ABB RAPID module: Module1.mod

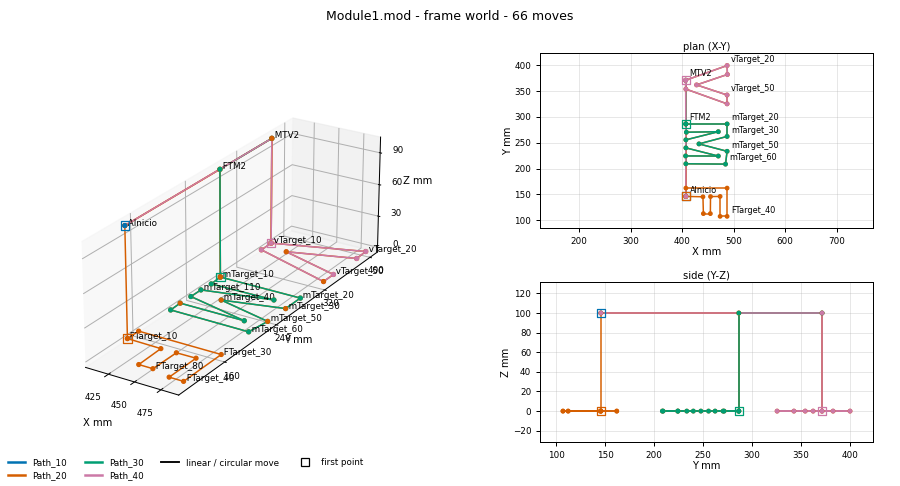
[picture p0: tool path of Module1.mod in frame world, 66 of 68 moves have a stored position in this frame; points joined in program order, loops and branches not executed]
MODULE Module1
	CONST robtarget AInicio:=[[0,-225.593,-100],[1,0,0,0],[0,0,0,0],[9E+09,9E+09,9E+09,9E+09,9E+09,9E+09]];
	CONST robtarget FTarget_10:=[[0,-225.593,0],[1,0,0,0],[0,0,0,0],[9E+09,9E+09,9E+09,9E+09,9E+09,9E+09]];
	CONST robtarget FTarget_20:=[[0,-209.44,0],[1,0,0,0],[0,0,0,0],[9E+09,9E+09,9E+09,9E+09,9E+09,9E+09]];
	CONST robtarget FTarget_30:=[[-80,-209.44,0],[1,0,0,0],[0,0,0,0],[9E+09,9E+09,9E+09,9E+09,9E+09,9E+09]];
	CONST robtarget FTarget_40:=[[-80,-264.284,0],[1,0,0,0],[0,0,0,0],[9E+09,9E+09,9E+09,9E+09,9E+09,9E+09]];
	CONST robtarget FTarget_50:=[[-66.466,-264.284,0],[1,0,0,0],[0,0,0,0],[9E+09,9E+09,9E+09,9E+09,9E+09,9E+09]];
	CONST robtarget FTarget_60:=[[-66.466,-225.593,0],[1,0,0,0],[0,0,0,0],[9E+09,9E+09,9E+09,9E+09,9E+09,9E+09]];
	CONST robtarget FTarget_70:=[[-47.849,-225.879,0],[1,0,0,0],[0,0,0,0],[9E+09,9E+09,9E+09,9E+09,9E+09,9E+09]];
	CONST robtarget FTarget_80:=[[-47.53,-258.99,0],[1,0,0,0],[0,0,0,0],[9E+09,9E+09,9E+09,9E+09,9E+09,9E+09]];
	CONST robtarget FTarget_90:=[[-33.997,-258.99,0],[1,0,0,0],[0,0,0,0],[9E+09,9E+09,9E+09,9E+09,9E+09,9E+09]];
	CONST robtarget FTarget_100:=[[-33.164,-226.306,0],[1,0,0,0],[0,0,0,0],[9E+09,9E+09,9E+09,9E+09,9E+09,9E+09]];
	CONST robtarget FTarget_110:=[[0,-225.593,0],[1,0,0,0],[0,0,0,0],[9E+09,9E+09,9E+09,9E+09,9E+09,9E+09]];
	CONST robtarget FTM1:=[[0,-225.593,-100],[1,0,0,0],[0,0,0,0],[9E+09,9E+09,9E+09,9E+09,9E+09,9E+09]];
	CONST robtarget FTM2:=[[0,-84.966,-100],[1,0,0,0],[0,0,0,0],[9E+09,9E+09,9E+09,9E+09,9E+09,9E+09]];
	CONST robtarget mTarget_10:=[[0,-84.966,0],[1,0,0,0],[0,0,0,0],[9E+09,9E+09,9E+09,9E+09,9E+09,9E+09]];
	CONST robtarget mTarget_20:=[[-80,-84.966,0],[1,0,0,0],[0,0,0,0],[9E+09,9E+09,9E+09,9E+09,9E+09,9E+09]];
	CONST robtarget mTarget_30:=[[-80,-109.14,0],[1,0,0,0],[0,0,0,0],[9E+09,9E+09,9E+09,9E+09,9E+09,9E+09]];
	CONST robtarget mTarget_40:=[[-25.429,-123.656,0],[1,0,0,0],[0,0,0,0],[9E+09,9E+09,9E+09,9E+09,9E+09,9E+09]];
	CONST robtarget mTarget_50:=[[-80,-138.008,0],[1,0,0,0],[0,0,0,0],[9E+09,9E+09,9E+09,9E+09,9E+09,9E+09]];
	CONST robtarget mTarget_60:=[[-76.954,-162.904,0],[1,0,0,0],[0,0,0,0],[9E+09,9E+09,9E+09,9E+09,9E+09,9E+09]];
	CONST robtarget mTarget_70:=[[0,-162.237,0],[1,0,0,0],[0,0,0,0],[9E+09,9E+09,9E+09,9E+09,9E+09,9E+09]];
	CONST robtarget mTarget_80:=[[0.53,-147.013,0],[1,0,0,0],[0,0,0,0],[9E+09,9E+09,9E+09,9E+09,9E+09,9E+09]];
	CONST robtarget mTarget_90:=[[-62.974,-147.23,0],[1,0,0,0],[0,0,0,0],[9E+09,9E+09,9E+09,9E+09,9E+09,9E+09]];
	CONST robtarget mTarget_100:=[[0,-131.35,0],[1,0,0,0],[0,0,0,0],[9E+09,9E+09,9E+09,9E+09,9E+09,9E+09]];
	CONST robtarget mTarget_110:=[[0,-115.798,0],[1,0,0,0],[0,0,0,0],[9E+09,9E+09,9E+09,9E+09,9E+09,9E+09]];
	CONST robtarget mTarget_120:=[[-62.974,-99.973,0],[1,0,0,0],[0,0,0,0],[9E+09,9E+09,9E+09,9E+09,9E+09,9E+09]];
	CONST robtarget mTarget_130:=[[-0.986,-101.003,0],[1,0,0,0],[0,0,0,0],[9E+09,9E+09,9E+09,9E+09,9E+09,9E+09]];
	CONST robtarget mTarget_140:=[[0,-84.966,0],[1,0,0,0],[0,0,0,0],[9E+09,9E+09,9E+09,9E+09,9E+09,9E+09]];
	CONST robtarget MTV1:=[[0,-84.966,-100],[1,0,0,0],[0,0,0,0],[9E+09,9E+09,9E+09,9E+09,9E+09,9E+09]];
	CONST robtarget MTV2:=[[0.326,-0.089,-100],[1,0,0,0],[0,0,0,0],[9E+09,9E+09,9E+09,9E+09,9E+09,9E+09]];
	CONST robtarget vTarget_10:=[[0.326,-0.089,0],[1,0,0,0],[0,0,0,0],[9E+09,9E+09,9E+09,9E+09,9E+09,9E+09]];
	CONST robtarget vTarget_20:=[[-80.066,28.469,0],[1,0,0,0],[0,0,0,0],[9E+09,9E+09,9E+09,9E+09,9E+09,9E+09]];
	CONST robtarget vTarget_30:=[[-80.616,11.146,0],[1,0,0,0],[0,0,0,0],[9E+09,9E+09,9E+09,9E+09,9E+09,9E+09]];
	CONST robtarget vTarget_40:=[[-20.791,-9.168,0],[1,0,0,0],[0,0,0,0],[9E+09,9E+09,9E+09,9E+09,9E+09,9E+09]];
	CONST robtarget vTarget_50:=[[-80,-28.758,0],[1,0,0,0],[0,0,0,0],[9E+09,9E+09,9E+09,9E+09,9E+09,9E+09]];
	CONST robtarget vTarget_60:=[[-80,-45.893,0],[1,0,0,0],[0,0,0,0],[9E+09,9E+09,9E+09,9E+09,9E+09,9E+09]];
	CONST robtarget vTarget_70:=[[0,-17.244,0],[1,0,0,0],[0,0,0,0],[9E+09,9E+09,9E+09,9E+09,9E+09,9E+09]];
	CONST robtarget vTarget_80:=[[0.326,-0.089,0],[1,0,0,0],[0,0,0,0],[9E+09,9E+09,9E+09,9E+09,9E+09,9E+09]];
	CONST robtarget vTarget_80_final:=[[0.326,-0.089,-100],[1,0,0,0],[0,0,0,0],[9E+09,9E+09,9E+09,9E+09,9E+09,9E+09]];
	CONST robtarget ZInicio:=[[0,-225.593,-100],[1,0,0,0],[0,0,0,0],[9E+09,9E+09,9E+09,9E+09,9E+09,9E+09]];
	CONST jointtarget HomePosition:=[[0,0,0,0,0,0],[9E+09,9E+09,9E+09,9E+09,9E+09,9E+09]];
	CONST jointtarget ChangeTool:=[[90.000002504,24.671787339,-34.427722191,-0.000016273,9.755934852,0.000016038],[9E+09,9E+09,9E+09,9E+09,9E+09,9E+09]];
    !***********************************************************
    !
    ! Módulo:  Module1
    !
    ! Descripción:
    !   <Introduzca la descripción aquí>
    !
    ! Autor: Administrador
    !
    ! Versión: 1.0
    !
    !***********************************************************


    !***********************************************************
    !
    ! Procedimiento Main
    !
    !   Este es el punto de entrada de su programa
    !
    !***********************************************************
    PROC main()
		Home1;
		WaitDI EntDI_1,1;
		SetDO SalDO_1,1;
		Path_10;
		Path_20;
		Home1;
		WaitDI EntDI_2,1;
		ToolChange;
		SetDO SalDO_1,0;
        !Añada aquí su código
    ENDPROC
	PROC Path_10()
	    MoveJ AInicio,v100,z10,Tooldata_MARCADOR\WObj:=Workobject_INICIALES;
	ENDPROC
	PROC Path_20()
	    MoveL FTarget_10,v100,z10,Tooldata_MARCADOR\WObj:=Workobject_INICIALES;
	    MoveL FTarget_20,v100,z10,Tooldata_MARCADOR\WObj:=Workobject_INICIALES;
	    MoveL FTarget_30,v100,z10,Tooldata_MARCADOR\WObj:=Workobject_INICIALES;
	    MoveL FTarget_40,v100,z10,Tooldata_MARCADOR\WObj:=Workobject_INICIALES;
	    MoveL FTarget_50,v100,z10,Tooldata_MARCADOR\WObj:=Workobject_INICIALES;
	    MoveL FTarget_60,v100,z10,Tooldata_MARCADOR\WObj:=Workobject_INICIALES;
	    MoveL FTarget_70,v100,z10,Tooldata_MARCADOR\WObj:=Workobject_INICIALES;
	    MoveL FTarget_80,v100,z10,Tooldata_MARCADOR\WObj:=Workobject_INICIALES;
	    MoveL FTarget_90,v100,z10,Tooldata_MARCADOR\WObj:=Workobject_INICIALES;
	    MoveL FTarget_100,v100,z10,Tooldata_MARCADOR\WObj:=Workobject_INICIALES;
	    MoveL FTarget_110,v100,z10,Tooldata_MARCADOR\WObj:=Workobject_INICIALES;
	    MoveL FTM1,v100,z10,Tooldata_MARCADOR\WObj:=Workobject_INICIALES;
	    MoveL FTM2,v100,z10,Tooldata_MARCADOR\WObj:=Workobject_INICIALES;
		MoveL mTarget_10,v100,z10,Tooldata_MARCADOR\WObj:=Workobject_INICIALES;
		MoveL mTarget_20,v100,z10,Tooldata_MARCADOR\WObj:=Workobject_INICIALES;
		MoveL mTarget_30,v100,z10,Tooldata_MARCADOR\WObj:=Workobject_INICIALES;
		MoveL mTarget_40,v100,z10,Tooldata_MARCADOR\WObj:=Workobject_INICIALES;
		MoveL mTarget_50,v100,z10,Tooldata_MARCADOR\WObj:=Workobject_INICIALES;
		MoveL mTarget_60,v100,z10,Tooldata_MARCADOR\WObj:=Workobject_INICIALES;
		MoveL mTarget_70,v100,z10,Tooldata_MARCADOR\WObj:=Workobject_INICIALES;
		MoveL mTarget_80,v100,z10,Tooldata_MARCADOR\WObj:=Workobject_INICIALES;
		MoveL mTarget_90,v100,z10,Tooldata_MARCADOR\WObj:=Workobject_INICIALES;
		MoveL mTarget_100,v100,z10,Tooldata_MARCADOR\WObj:=Workobject_INICIALES;
		MoveL mTarget_110,v100,z10,Tooldata_MARCADOR\WObj:=Workobject_INICIALES;
		MoveL mTarget_120,v100,z10,Tooldata_MARCADOR\WObj:=Workobject_INICIALES;
		MoveL mTarget_130,v100,z10,Tooldata_MARCADOR\WObj:=Workobject_INICIALES;
		MoveL mTarget_140,v100,z10,Tooldata_MARCADOR\WObj:=Workobject_INICIALES;
		MoveL MTV1,v100,z10,Tooldata_MARCADOR\WObj:=Workobject_INICIALES;
		MoveL MTV2,v100,z10,Tooldata_MARCADOR\WObj:=Workobject_INICIALES;
		MoveL vTarget_10,v100,z10,Tooldata_MARCADOR\WObj:=Workobject_INICIALES;
		MoveL vTarget_20,v100,z10,Tooldata_MARCADOR\WObj:=Workobject_INICIALES;
		MoveL vTarget_30,v100,z10,Tooldata_MARCADOR\WObj:=Workobject_INICIALES;
		MoveL vTarget_40,v100,z10,Tooldata_MARCADOR\WObj:=Workobject_INICIALES;
		MoveL vTarget_50,v100,z10,Tooldata_MARCADOR\WObj:=Workobject_INICIALES;
		MoveL vTarget_60,v100,z10,Tooldata_MARCADOR\WObj:=Workobject_INICIALES;
		MoveL vTarget_70,v100,z10,Tooldata_MARCADOR\WObj:=Workobject_INICIALES;
		MoveL vTarget_80,v100,z10,Tooldata_MARCADOR\WObj:=Workobject_INICIALES;
		MoveL vTarget_80_final,v100,z10,Tooldata_MARCADOR\WObj:=Workobject_INICIALES;
		MoveL ZInicio,v100,z10,Tooldata_MARCADOR\WObj:=Workobject_INICIALES;
	ENDPROC
	PROC Path_30()
	    MoveL mTarget_10,v100,z10,Tooldata_MARCADOR\WObj:=Workobject_INICIALES;
	    MoveL mTarget_20,v100,z10,Tooldata_MARCADOR\WObj:=Workobject_INICIALES;
	    MoveL mTarget_30,v100,z10,Tooldata_MARCADOR\WObj:=Workobject_INICIALES;
	    MoveL mTarget_40,v100,z10,Tooldata_MARCADOR\WObj:=Workobject_INICIALES;
	    MoveL mTarget_50,v100,z10,Tooldata_MARCADOR\WObj:=Workobject_INICIALES;
	    MoveL mTarget_60,v100,z10,Tooldata_MARCADOR\WObj:=Workobject_INICIALES;
	    MoveL mTarget_70,v100,z10,Tooldata_MARCADOR\WObj:=Workobject_INICIALES;
	    MoveL mTarget_80,v100,z10,Tooldata_MARCADOR\WObj:=Workobject_INICIALES;
	    MoveL mTarget_90,v100,z10,Tooldata_MARCADOR\WObj:=Workobject_INICIALES;
	    MoveL mTarget_100,v100,z10,Tooldata_MARCADOR\WObj:=Workobject_INICIALES;
	    MoveL mTarget_110,v100,z10,Tooldata_MARCADOR\WObj:=Workobject_INICIALES;
	    MoveL mTarget_120,v100,z10,Tooldata_MARCADOR\WObj:=Workobject_INICIALES;
	    MoveL mTarget_130,v100,z10,Tooldata_MARCADOR\WObj:=Workobject_INICIALES;
	    MoveL mTarget_140,v100,z10,Tooldata_MARCADOR\WObj:=Workobject_INICIALES;
	    MoveL MTV1,v100,z10,Tooldata_MARCADOR\WObj:=Workobject_INICIALES;
	    MoveL MTV2,v100,z10,Tooldata_MARCADOR\WObj:=Workobject_INICIALES;
	ENDPROC
	PROC Path_40()
	    MoveL vTarget_10,v100,z10,Tooldata_MARCADOR\WObj:=Workobject_INICIALES;
	    MoveL vTarget_20,v100,z10,Tooldata_MARCADOR\WObj:=Workobject_INICIALES;
	    MoveL vTarget_30,v100,z10,Tooldata_MARCADOR\WObj:=Workobject_INICIALES;
	    MoveL vTarget_40,v100,z10,Tooldata_MARCADOR\WObj:=Workobject_INICIALES;
	    MoveL vTarget_50,v100,z10,Tooldata_MARCADOR\WObj:=Workobject_INICIALES;
	    MoveL vTarget_60,v100,z10,Tooldata_MARCADOR\WObj:=Workobject_INICIALES;
	    MoveL vTarget_70,v100,z10,Tooldata_MARCADOR\WObj:=Workobject_INICIALES;
	    MoveL vTarget_80,v100,z10,Tooldata_MARCADOR\WObj:=Workobject_INICIALES;
	    MoveL vTarget_80_final,v100,z10,Tooldata_MARCADOR\WObj:=Workobject_INICIALES;
	    MoveL ZInicio,v100,z10,Tooldata_MARCADOR\WObj:=Workobject_INICIALES;
	ENDPROC
	PROC Home1()
	    MoveAbsJ HomePosition,v100,z10,Tooldata_MARCADOR\WObj:=Workobject_INICIALES;
	ENDPROC
	PROC ToolChange()
	    MoveAbsJ ChangeTool,v50,z10,Tooldata_MARCADOR\WObj:=Workobject_INICIALES;
	ENDPROC
ENDMODULE
